{attribute addProperty BoxType "EK1122-0000-0018"}
{attribute addProperty Id "Beckhoff_EP4xxxsub_EK1100EK1100_179A0949162A_0001_EP4174_0002_0016EP4174_9786CACB14518.125A_0002_EP4174_0002_0017EP4174_9786CACB14518.125A_0003_EP4174_0002_0018EP4174_9786CACB14518.125A_0004_EP4174_0002_0019EP4174_9786CACB14518.125A_0005_EP4314_1002_0016EP4314_D38CD2FF21026.25A_0006_EP4374_0002_0016EP4374_74CDCD2417822.25A_0007_EP4374_0002_0017EP4374_6989BFFB17822.25A_0008_EP4374_0002_0018EP4374_6989BFFB17822.25A_0009_EP4374_0002_0019EP4374_6989BFFB17822.25A_0010_EP4378_1022_0017EP4378_B0B1C4E640250.25"}
{attribute addProperty CRC "3143908699"}
{attribute addProperty SizeInBites "1920"}
{attribute addProperty SizeInBytes "240"}
TYPE Beckhoff_EP4xxxEK1122_BB643D5B EXTENDS EK1122_179A0949 :
STRUCT
	{attribute addProperty Name "Beckhoff_EP4xxxsub_EK1100"}
	Beckhoff_EP4xxxsub_EK1100 : EK1100_179A0949;
	{attribute addProperty Name "A_0001_EP4174_0002_0016"}
	A_0001_EP4174_0002_0016 : EP4174_9786CACB;
	{attribute addProperty Name "A_0002_EP4174_0002_0017"}
	A_0002_EP4174_0002_0017 : EP4174_9786CACB;
	{attribute addProperty Name "A_0003_EP4174_0002_0018"}
	A_0003_EP4174_0002_0018 : EP4174_9786CACB;
	{attribute addProperty Name "A_0004_EP4174_0002_0019"}
	A_0004_EP4174_0002_0019 : EP4174_9786CACB;
	{attribute addProperty Name "A_0005_EP4314_1002_0016"}
	A_0005_EP4314_1002_0016 : EP4314_D38CD2FF;
	{attribute addProperty Name "A_0006_EP4374_0002_0016"}
	A_0006_EP4374_0002_0016 : EP4374_74CDCD24;
	{attribute addProperty Name "A_0007_EP4374_0002_0017"}
	A_0007_EP4374_0002_0017 : EP4374_6989BFFB;
	{attribute addProperty Name "A_0008_EP4374_0002_0018"}
	A_0008_EP4374_0002_0018 : EP4374_6989BFFB;
	{attribute addProperty Name "A_0009_EP4374_0002_0019"}
	A_0009_EP4374_0002_0019 : EP4374_6989BFFB;
	{attribute addProperty Name "A_0010_EP4378_1022_0017"}
	A_0010_EP4378_1022_0017 : EP4378_B0B1C4E6;
END_STRUCT
END_TYPE

(* stored: Version 1.2.0.0, ProductVersion 3.1.4024.9
   DUT Beckhoff_EP4xxxEK1122_BB643D5B: Id {6eff3106-c640-44f5-9307-41d6ec21a080} *)
